PROGRAM PRG_MR1K4_SOMS
VAR
    // M1K4 Flow Press Sensors
    {attribute 'TcLinkTo' := '.fbFlow_1.iRaw := TIIB[EL3054_M1K4_FWM_PRSM]^AI Standard Channel 1^Value;
                                 .fbFlow_2.iRaw := TIIB[EL3054_M1K4_FWM_PRSM]^AI Standard Channel 2^Value;
                              .fbPress_1.iRaw := TIIB[EL3054_M1K4_FWM_PRSM]^AI Standard Channel 3^Value
    '}
    {attribute 'pytmc' := '
        pv: MR1K4:SOMS
    '}
    fbCoolingPanel : FB_Axilon_Cooling_2f1p;
    {attribute 'TcLinkTo' := 'TIIB[EP2008-0001_M1K4_VCV]^Channel 1^Output'}
    {attribute 'pytmc' := '
        pv: MR1K4:SOMS:VCV
        io: io
        field: ZNAM OFF
        field: ONAM ON
    '}
    bActivateVarCool AT %Q* : BOOL;
END_VAR

fbCoolingPanel();

END_PROGRAM

(* stored: Version 1.1.0.1, ProductVersion 3.1.4024.12
   POU PRG_MR1K4_SOMS: Id {b187bbdf-2876-4f23-8b37-07bf843b3938}, SpecialFunc None *)
